FUNCTION_BLOCK ABSTRACT FB_Base IMPLEMENTS ITF_Base
VAR
	_Definition				: ST_BaseDefinition;
	_EnableManualControl	: BOOL;
END_VAR

PROPERTY Definition : REFERENCE TO ST_BaseDefinition
GET
Definition REF= _Definition;
END_GET
END_PROPERTY

PROPERTY EnableManualControl : BOOL
SET
_EnableManualControl := EnableManualControl;
END_SET
END_PROPERTY

END_FUNCTION_BLOCK

(* stored: Version 1.1.0.1
   POU FB_Base: Id {1b877d1c-c148-4ce1-b504-f1a684f4690b}, SpecialFunc None
   Property Definition: Id {b6a8add8-928c-44fd-95f2-a7123022e2b1}
   Get Get: Id {79215c66-6435-4348-887a-de976332b211}
   Property EnableManualControl: Id {878b68fe-e504-47d7-a7db-91ff55dbb844}
   Set Set: Id {02d5433a-364f-43db-bf26-31ce824317bc} *)
